(* PLC project Methods Example.project, CODESYS CODESYS V3.5 SP20 Patch 1 *)
(* stored: creationDateTime 2025-05-26T20:50:46.0607646, modificationDateTime 2025-05-23T12:04:24.0034929 *)

PROGRAM Main
  VAR_INPUT
    MotorA : Motor;
    methodHasCompleted : BOOL;
  END_VAR

                    
// Call a method and get the return value

methodHasCompleted := MotorA.Start();
                  
END_PROGRAM

FUNCTION_BLOCK Motor
  VAR
    MotorRunOutput : BOOL;
  END_VAR

                    
                  

METHOD Start : BOOL
                          
// Check motor is ok to start then...

MotorRunOutput := TRUE;

// Return a value
Start := TRUE;
                        
END_METHOD

METHOD Stop : BOOL
                          
// Check motor is ok to stop then...

MotorRunOutput := FALSE;
                        
END_METHOD
END_FUNCTION_BLOCK

CONFIGURATION Device
  RESOURCE Application ON PLC
    TASK MainTask(INTERVAL := T#20ms, PRIORITY := 1);
    PROGRAM Main WITH MainTask : Main;
  END_RESOURCE
END_CONFIGURATION
